ABB RobotStudio station: convertracking.rsstn

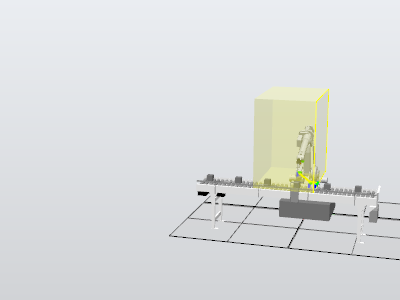
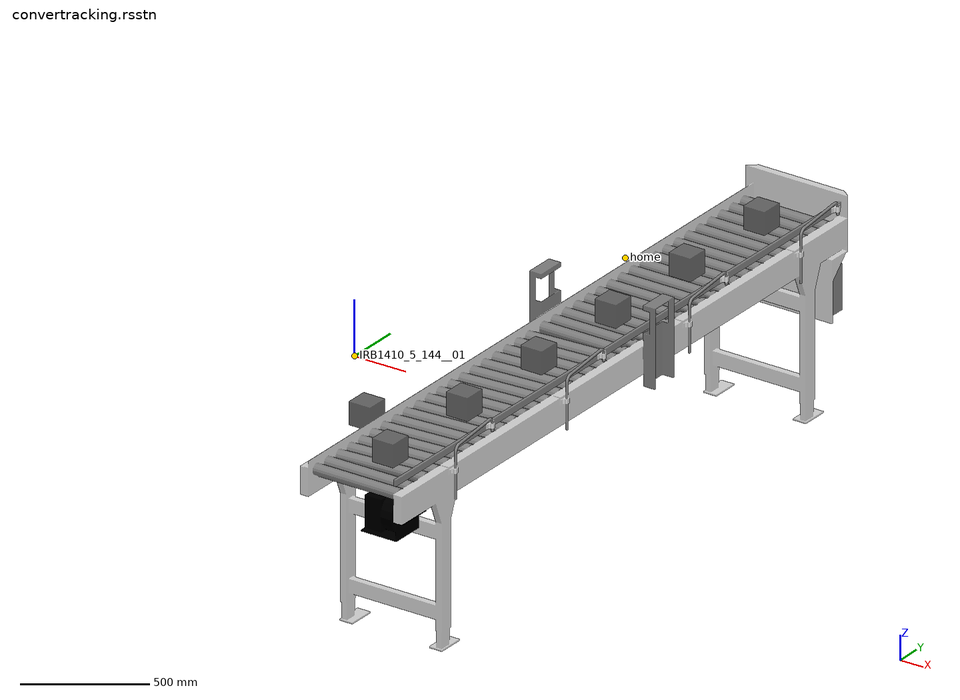
[picture v1: parts stored in the station drawn from their meshes, with robot base, taught points and paths (robot models come from the ABB library and are not in the file)]
Station project 2 (saved by RobotStudio 22.3.10141.1)
Controller Controller3, task T_ROB1: task frame (RAPID world) sits at (181.67, 237.14, 303.24) mm in the station
Controller Controller3
  mechanical unit ROB_1: IRB1410_5_144__01, 6 joints, base frame (-153.04, -239.98, 0) mm
  mechanical unit CNV1: ?, 1 joints, base frame (818.33, 62.86, 496.76) mm, rotated rx 0 ry 0 rz -90 deg
Layout (positions relative to the parent item):
  - IRB1410_5_144__01 [mechanism, from Robots\IRB1410_5_144_G_01.rslib] at (28.62, -2.83, 303.24) mm; joint values [0.0075, 0.2384, 0.3018, -0.0297, 0.2219, 0.0327] (rad or m)
  - concrete [part, from Dispencing\Concrete.rslib] at (-450, -450, 0) mm
  - MyTool_2 [mechanism, from Training Objects\myTool.rslib] at (1117.02, 4.82, 1219.33) mm, rotated rx -180 ry 60 rz -180 deg
  - Conveyor [conveyor]
    - 400_guide [part] at (1000, 1300, 0) mm, rotated rx 0 ry 0 rz -90 deg, size 3033 x 590 x 945 mm
    - Part_2 [part], size 100 x 100 x 100 mm
    - ConveyorObject_6 [conveyorobject] at (1000, -1458.09, 800) mm, rotated rx 0 ry 0 rz -90 deg
      - Part_2 [part] at (0, 200, 0) mm, size 100 x 100 x 100 mm
    - ConveyorObject_7 [conveyorobject] at (1000, -958.09, 800) mm, rotated rx 0 ry 0 rz -90 deg
      - Part_2 [part] at (0, 200, 0) mm, size 100 x 100 x 100 mm
    - ConveyorObject_8 [conveyorobject] at (1000, -458.09, 800) mm, rotated rx 0 ry 0 rz -90 deg
      - Part_2 [part] at (0, 200, 0) mm, size 100 x 100 x 100 mm
    - ConveyorObject_9 [conveyorobject] at (1000, 41.91, 800) mm, rotated rx 0 ry 0 rz -90 deg
      - Part_2 [part] at (0, 200, 0) mm, size 100 x 100 x 100 mm
    - ConveyorObject_10 [conveyorobject] at (1000, 541.91, 800) mm, rotated rx 0 ry 0 rz -90 deg
      - Part_2 [part] at (0, 200, 0) mm, size 100 x 100 x 100 mm
    - ConveyorObject_7 [conveyorobject] at (1000, 1041.91, 800) mm, rotated rx 0 ry 0 rz -90 deg
      - Part_2 [part] at (0, 200, 0) mm, size 100 x 100 x 100 mm
Attachment: MyTool_2 is attached to IRB1410_5_144__01 / Link6
Conveyor tracking Connection: unit CNV1, TravelOffset=1, QueueTrackDistance=0, StartWindowWidth=1, SyncSeparation=0.1, CountsPerMeter=10000
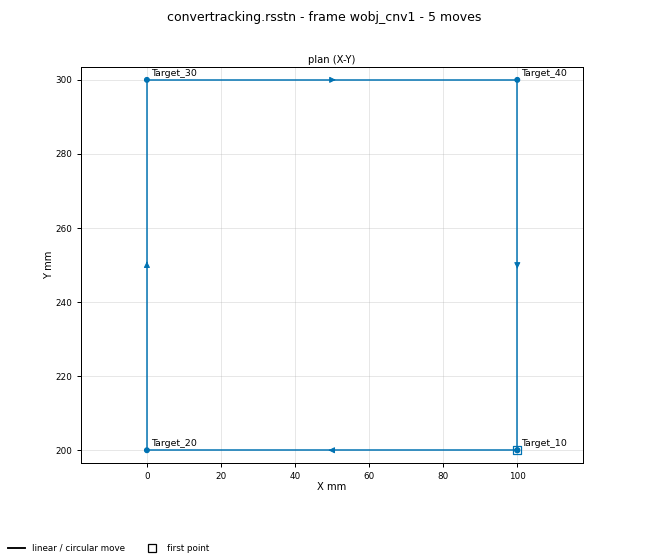
[picture p0: tool path of convertracking.rsstn in frame wobj_cnv1, 5 of 7 moves have a stored position in this frame; points joined in program order, loops and branches not executed]
Targets, tools, work objects and paths stored in the station, written as RAPID:
! task T_ROB1
MODULE CalibData
  PERS tooldata MyTool:=[TRUE,[[31.792631019,0,229.638935148],[0.945518576,0,0.325568154,0]],[1,[0,0,1],[1,0,0,0],0,0,0]];
  TASK PERS wobjdata wobj_cnv1:=[FALSE,FALSE,"CNV1",[[0,-163.551498115,-7.237041676],[0.707106781,0,0,0.707106781]],[[0,0,0],[1,0,0,0]]];
ENDMODULE

! task T_ROB1
MODULE Module1
  CONST robtarget home:=[[1118.333027957,-232.320473322,773.743955998],[0.190808342,-0.00000005,0.98162731,-0.000000041],[-1,0,-1,0],[9E+09,9E+09,9E+09,9E+09,9E+09,0]];
  CONST robtarget Target_10:=[[100.000035537,199.999648621,99.999984957],[0.134921749,-0.694115377,0.694115332,0.134921723],[0,0,-1,0],[9E+09,9E+09,9E+09,9E+09,9E+09,0]];
  CONST robtarget Target_20:=[[0.000038103,199.999656539,99.999995261],[0.134921696,-0.694115396,0.694115338,0.134921648],[0,0,-1,0],[9E+09,9E+09,9E+09,9E+09,9E+09,0]];
  CONST robtarget Target_30:=[[0.000038533,299.999686448,99.999996469],[0.134921708,-0.6941154,0.694115332,0.134921641],[0,1,-1,0],[9E+09,9E+09,9E+09,9E+09,9E+09,0]];
  CONST robtarget Target_40:=[[100.000044416,299.999686585,99.999998357],[0.134921713,-0.694115404,0.694115329,0.134921631],[0,0,-1,0],[9E+09,9E+09,9E+09,9E+09,9E+09,0]];
  PROC Path_10()
    ActUnit CNV1;
    MoveL home,v1000,z100,MyTool\WObj:=wobj0;
    WaitWObj wobj_cnv1;
    MoveL Target_10,v1000,z100,MyTool\WObj:=wobj_cnv1;
    MoveL Target_20,v1000,z100,MyTool\WObj:=wobj_cnv1;
    MoveL Target_30,v1000,z100,MyTool\WObj:=wobj_cnv1;
    MoveL Target_40,v1000,z100,MyTool\WObj:=wobj_cnv1;
    MoveL Target_10,v1000,z100,MyTool\WObj:=wobj_cnv1;
    MoveL home,v1000,z100,MyTool\WObj:=wobj0;
    WaitTime 1;
    DropWObj wobj_cnv1;
  ENDPROC
ENDMODULE

